FUNCTION_BLOCK F_FT_LIMIT (* Basic Function Block Type *)
  (* Standard: 61499-2 *)
  (* Version 0.0, 2013-10-19, 4DIAC-IDE, 4DIAC-Consortium *)
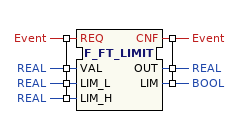
  EVENT_INPUT
    REQ WITH LIM_L, VAL, LIM_H; (* Normal Execution Request *)
  END_EVENT
  EVENT_OUTPUT
    CNF WITH OUT, LIM; (* Execution Confirmation *)
  END_EVENT
  VAR_INPUT
    VAL : REAL;
    LIM_L : REAL := -1.0E38; (* Input event qualifier *)
    LIM_H : REAL := 1.0E38;
  END_VAR
  VAR_OUTPUT
    OUT : REAL; (* Output event qualifier *)
    LIM : BOOL;
  END_VAR
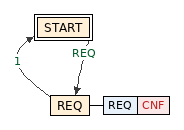
  EC_STATES
    START; (* Initial State *)
    REQ : REQ -> CNF; (* Normal execution *)
  END_STATES
  EC_TRANSITIONS
    START TO REQ := REQ;
    REQ TO START := 1;
  END_TRANSITIONS
  ALGORITHM REQ IN ST: (* Normally executed algorithm *)
OUT := VAL;

(* limit the output *)
IF OUT < LIM_L THEN
	LIM := TRUE;
	OUT := LIM_L;
ELSIF OUT > LIM_H THEN
	LIM := TRUE;
	OUT := LIM_H;
ELSE
	LIM := FALSE;
END_IF;
  END_ALGORITHM
END_FUNCTION_BLOCK
